FUNCTION_BLOCK FB_RobotComms
VAR
	timWatchDogON: TON;
	timWatchDogOff: TON;
	timMotorsOnFault: TON;
	timMotorsOffFault: TON;
	qMotorsOffFault: BOOL;
	timRunningFault: TON;
	timRunningStopFault: TON;
	tRunRoutine: BOOL;
	timRoutineRunFault: TON;
	tRoutineValMismatch: BOOL;
	timRoutineValMismatchFault: TON;
	qRoutineMismatch: BOOL;
	tRoutineValNotZero: BOOL;
	tRoutineComplete: BOOL;
	tCheckForEndPose: BOOL;
	tCheckForEndPosn: BOOL;
	timFakeRunSignal: TON;
END_VAR

VAR_INPUT
//	iStationPowerOn:BOOL;
//	iStationManualMode:BOOL;
//	iStationAutoCycling:BOOL;
END_VAR
	
VAR_IN_OUT
	iqRobotData:structRobot;
	station:typeStation; //data relating to the entire station
	
END_VAR

VAR_OUTPUT
	qWatchdogFault: BOOL;
	qMotorsOnFault: BOOL;
	qProgramRunFault: BOOL;
	qRoutinePoseFault: BOOL;
	qCollisionFault:BOOL;
END_VAR

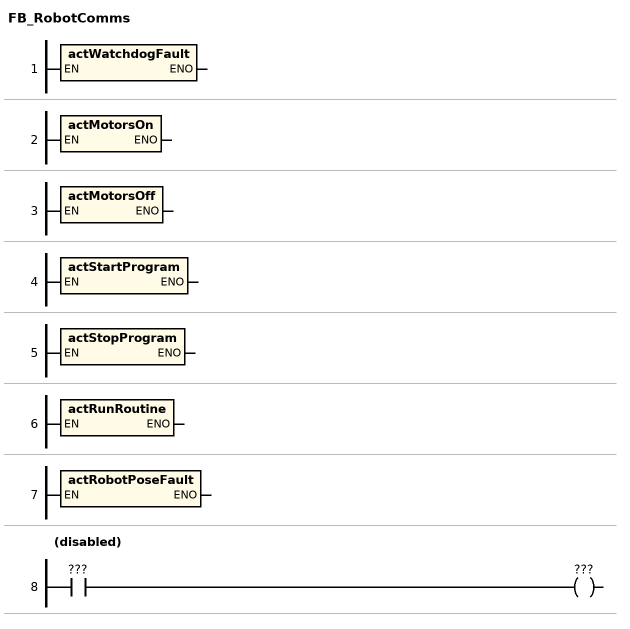
// NETWORK 1
actWatchdogFault();

// NETWORK 2
actMotorsOn();

// NETWORK 3
actMotorsOff();

// NETWORK 4
actStartProgram();

// NETWORK 5
actStopProgram();

// NETWORK 6
actRunRoutine();

// NETWORK 7
actRobotPoseFault();

// NETWORK 8 (disabled)
// ??? := ???;

ACTION actCollision:
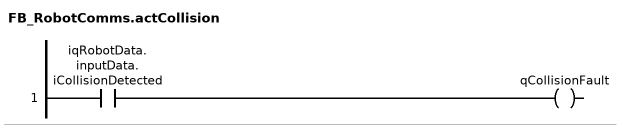
// NETWORK 1
qCollisionFault := iqRobotData.inputData.iCollisionDetected;
END_ACTION

ACTION actMotorsOff:
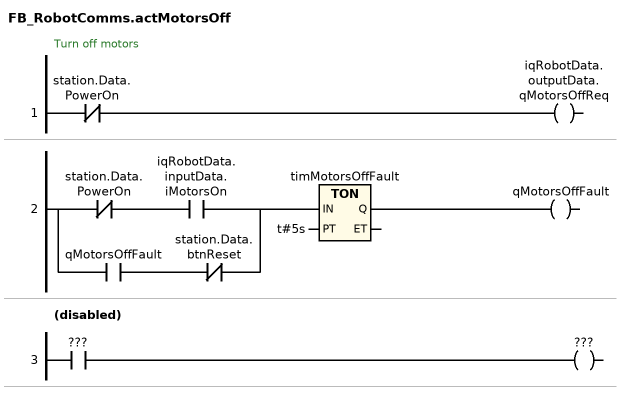
// NETWORK 1
// Turn off motors
iqRobotData.outputData.qMotorsOffReq := NOT station.Data.PowerOn;

// NETWORK 2
timMotorsOffFault(IN := NOT station.Data.PowerOn AND iqRobotData.inputData.iMotorsOn OR qMotorsOffFault AND NOT station.Data.btnReset, PT := t#5s); // TON
qMotorsOffFault := timMotorsOffFault.Q;

// NETWORK 3 (disabled)
// ??? := ???;
END_ACTION

ACTION actMotorsOn:
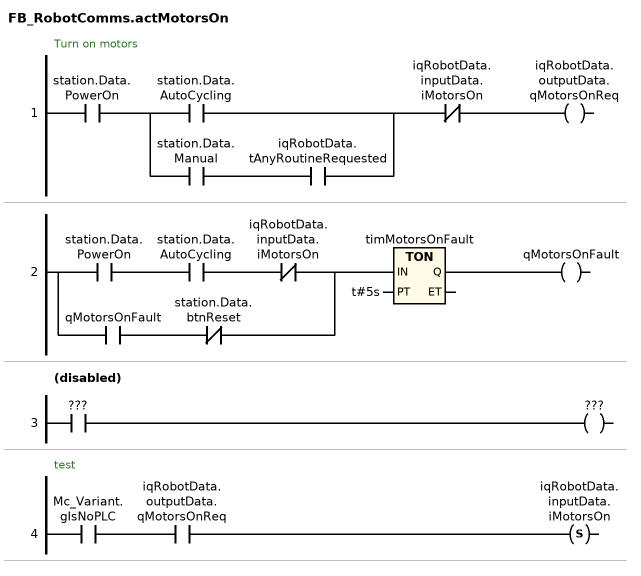
// NETWORK 1
// Turn on motors
iqRobotData.outputData.qMotorsOnReq := station.Data.PowerOn AND (station.Data.AutoCycling OR station.Data.Manual AND iqRobotData.tAnyRoutineRequested) AND NOT iqRobotData.inputData.iMotorsOn;

// NETWORK 2
timMotorsOnFault(IN := station.Data.PowerOn AND station.Data.AutoCycling AND NOT iqRobotData.inputData.iMotorsOn OR qMotorsOnFault AND NOT station.Data.btnReset, PT := t#5s); // TON
qMotorsOnFault := timMotorsOnFault.Q;

// NETWORK 3 (disabled)
// ??? := ???;

// NETWORK 4
// test
iqRobotData.inputData.iMotorsOn S= Mc_Variant.gIsNoPLC AND iqRobotData.outputData.qMotorsOnReq;
END_ACTION

ACTION actRobotPoseFault:
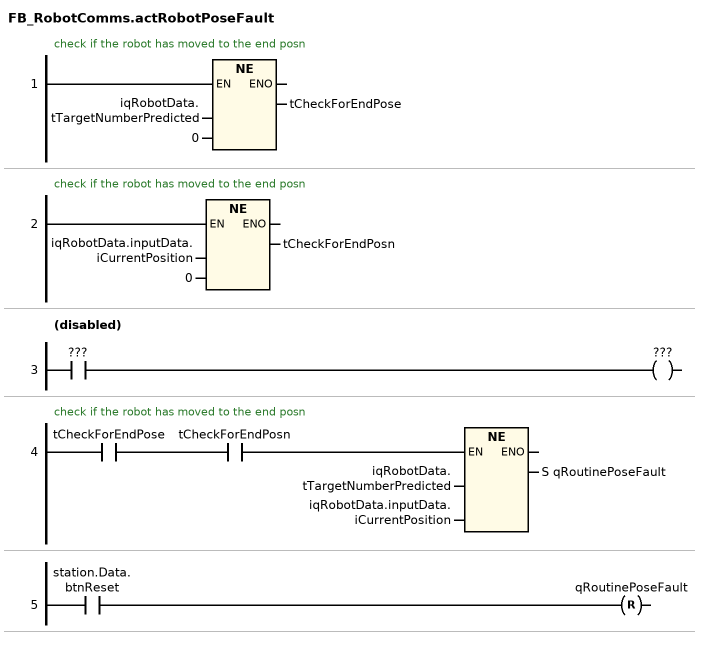
// NETWORK 1
// check if the robot has moved to the end posn
tCheckForEndPose := iqRobotData.tTargetNumberPredicted <> 0;

// NETWORK 2
// check if the robot has moved to the end posn
tCheckForEndPosn := iqRobotData.inputData.iCurrentPosition <> 0;

// NETWORK 3 (disabled)
// ??? := ???;

// NETWORK 4
// check if the robot has moved to the end posn
IF tCheckForEndPose AND tCheckForEndPosn THEN
    qRoutinePoseFault S= iqRobotData.tTargetNumberPredicted <> iqRobotData.inputData.iCurrentPosition;
END_IF

// NETWORK 5
qRoutinePoseFault R= station.Data.btnReset;
END_ACTION

ACTION actRunRoutine:
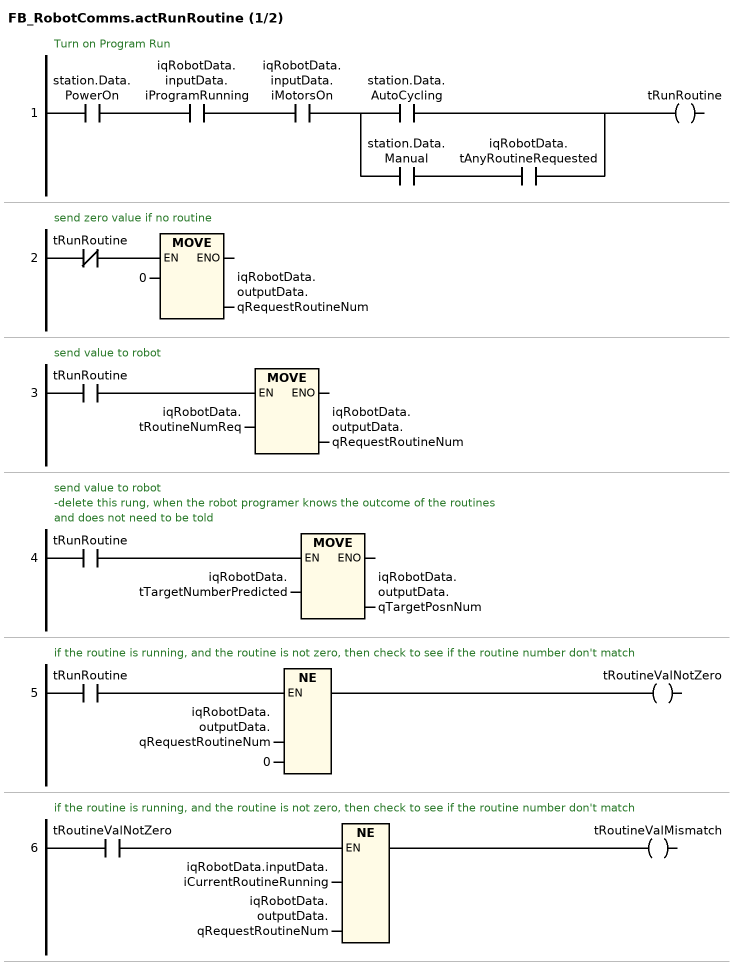
// NETWORK 1
// Turn on Program Run
tRunRoutine := station.Data.PowerOn AND iqRobotData.inputData.iProgramRunning AND iqRobotData.inputData.iMotorsOn AND (station.Data.AutoCycling OR station.Data.Manual AND iqRobotData.tAnyRoutineRequested);

// NETWORK 2
// send zero value if no routine
IF NOT tRunRoutine THEN iqRobotData.outputData.qRequestRoutineNum := 0; END_IF

// NETWORK 3
// send value to robot
IF tRunRoutine THEN iqRobotData.outputData.qRequestRoutineNum := iqRobotData.tRoutineNumReq; END_IF

// NETWORK 4
// send value to robot
// -delete this rung, when the robot programer knows the outcome of the routines
// and does not need to be told
IF tRunRoutine THEN iqRobotData.outputData.qTargetPosnNum := iqRobotData.tTargetNumberPredicted; END_IF

// NETWORK 5
// if the routine is running, and the routine is not zero, then check to see if the routine number don't match
tRoutineValNotZero := tRunRoutine AND iqRobotData.outputData.qRequestRoutineNum <> 0;

// NETWORK 6
// if the routine is running, and the routine is not zero, then check to see if the routine number don't match
tRoutineValMismatch := tRoutineValNotZero AND iqRobotData.inputData.iCurrentRoutineRunning <> iqRobotData.outputData.qRequestRoutineNum;

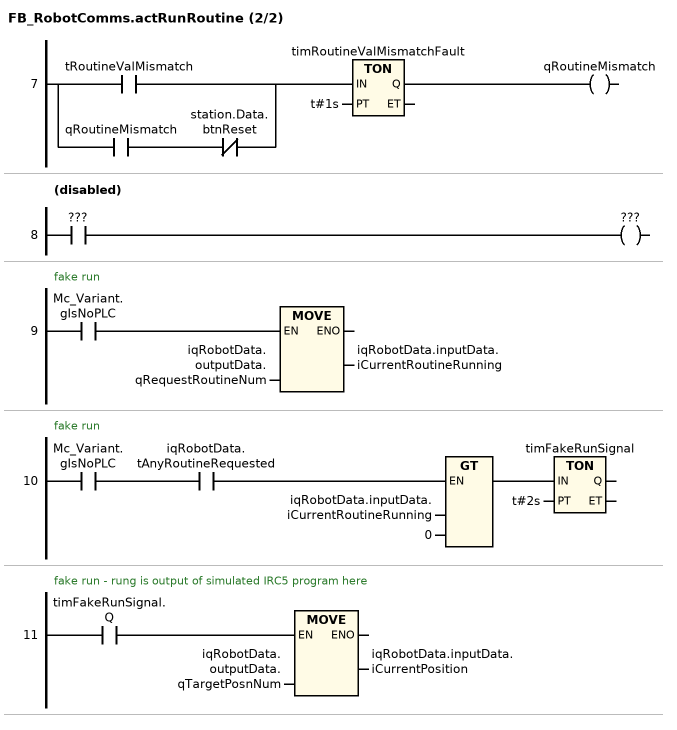
// NETWORK 7
timRoutineValMismatchFault(IN := tRoutineValMismatch OR qRoutineMismatch AND NOT station.Data.btnReset, PT := t#1s); // TON
qRoutineMismatch := timRoutineValMismatchFault.Q;

// NETWORK 8 (disabled)
// ??? := ???;

// NETWORK 9
// fake run
IF Mc_Variant.gIsNoPLC THEN
    iqRobotData.inputData.iCurrentRoutineRunning := iqRobotData.outputData.qRequestRoutineNum;
END_IF

// NETWORK 10
// fake run
timFakeRunSignal(IN := Mc_Variant.gIsNoPLC AND iqRobotData.tAnyRoutineRequested AND iqRobotData.inputData.iCurrentRoutineRunning > 0, PT := t#2s); // TON

// NETWORK 11
// fake run - rung is output of simulated IRC5 program here
IF timFakeRunSignal.Q THEN iqRobotData.inputData.iCurrentPosition := iqRobotData.outputData.qTargetPosnNum; END_IF
END_ACTION

ACTION actStartProgram:
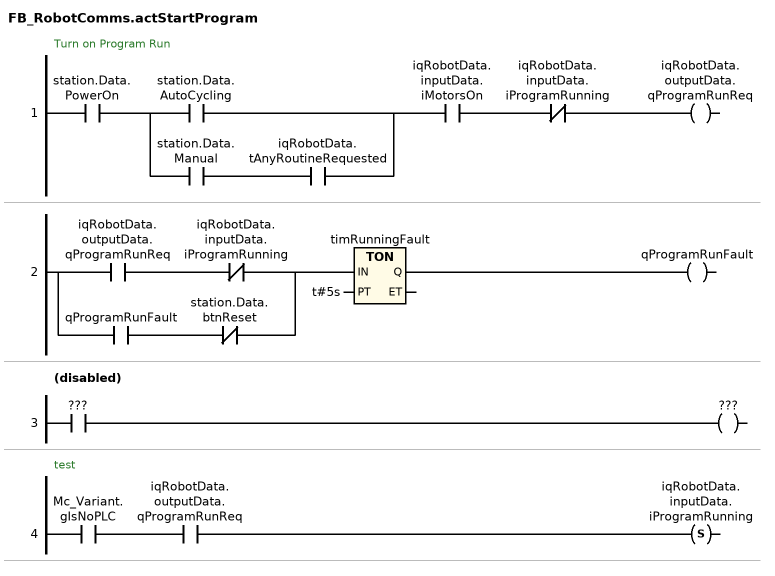
// NETWORK 1
// Turn on Program Run
iqRobotData.outputData.qProgramRunReq := station.Data.PowerOn AND (station.Data.AutoCycling OR station.Data.Manual AND iqRobotData.tAnyRoutineRequested) AND iqRobotData.inputData.iMotorsOn AND NOT iqRobotData.inputData.iProgramRunning;

// NETWORK 2
timRunningFault(IN := iqRobotData.outputData.qProgramRunReq AND NOT iqRobotData.inputData.iProgramRunning OR qProgramRunFault AND NOT station.Data.btnReset, PT := t#5s); // TON
qProgramRunFault := timRunningFault.Q;

// NETWORK 3 (disabled)
// ??? := ???;

// NETWORK 4
// test
iqRobotData.inputData.iProgramRunning S= Mc_Variant.gIsNoPLC AND iqRobotData.outputData.qProgramRunReq;
END_ACTION

ACTION actStopProgram:
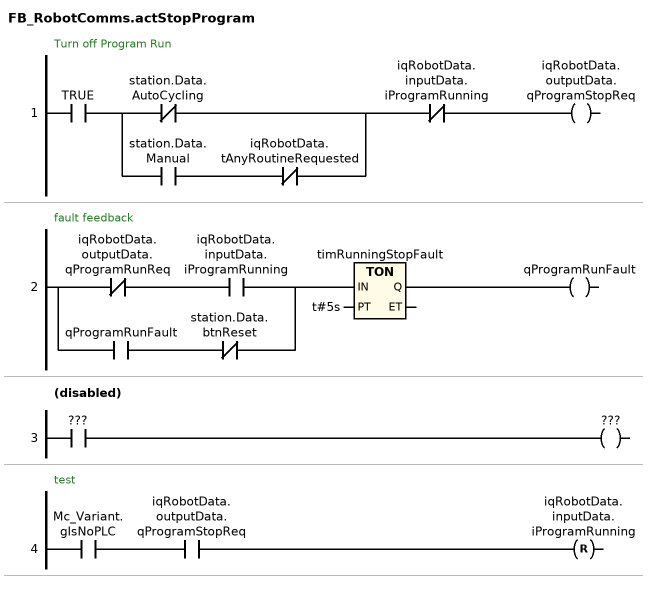
// NETWORK 1
// Turn off Program Run
iqRobotData.outputData.qProgramStopReq := TRUE AND (NOT station.Data.AutoCycling OR station.Data.Manual AND NOT iqRobotData.tAnyRoutineRequested) AND NOT iqRobotData.inputData.iProgramRunning;

// NETWORK 2
// fault feedback
timRunningStopFault(IN := NOT iqRobotData.outputData.qProgramRunReq AND iqRobotData.inputData.iProgramRunning OR qProgramRunFault AND NOT station.Data.btnReset, PT := t#5s); // TON
qProgramRunFault := timRunningStopFault.Q;

// NETWORK 3 (disabled)
// ??? := ???;

// NETWORK 4
// test
iqRobotData.inputData.iProgramRunning R= Mc_Variant.gIsNoPLC AND iqRobotData.outputData.qProgramStopReq;
END_ACTION

ACTION actWatchdogFault:
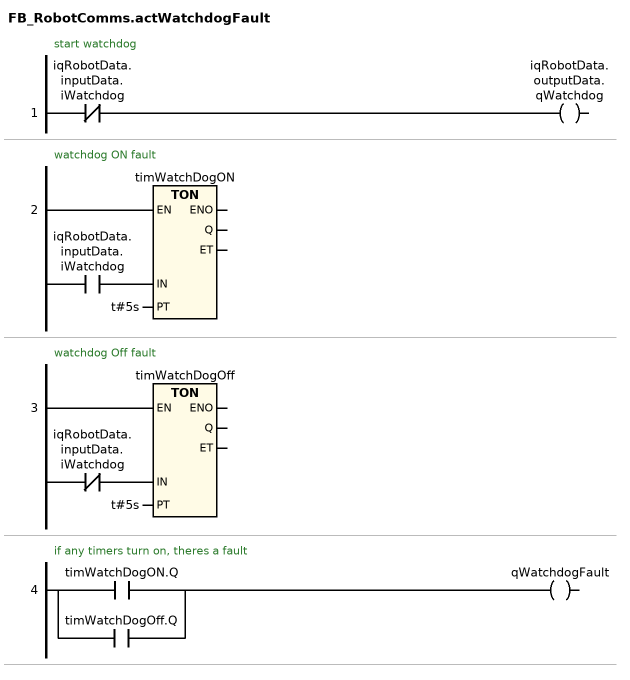
// NETWORK 1
// start watchdog
iqRobotData.outputData.qWatchdog := NOT iqRobotData.inputData.iWatchdog;

// NETWORK 2
// watchdog ON fault
timWatchDogON(IN := iqRobotData.inputData.iWatchdog, PT := t#5s); // TON

// NETWORK 3
// watchdog Off fault
timWatchDogOff(IN := NOT iqRobotData.inputData.iWatchdog, PT := t#5s); // TON

// NETWORK 4
// if any timers turn on, theres a fault
qWatchdogFault := timWatchDogON.Q OR timWatchDogOff.Q;
END_ACTION

END_FUNCTION_BLOCK

(* stored: Version 1.1.0.1, ProductVersion 3.1.4024.11
   POU FB_RobotComms: Id {38d8d4f8-9dcc-4020-a9d8-b9eb8bd54575}, SpecialFunc None
   Action actCollision: Id {ad7d7a71-11d1-4d2a-9400-4cf98c8d3ece}
   Action actMotorsOff: Id {3aae55ed-d4e0-4023-9d06-b2d9a8891dff}
   Action actMotorsOn: Id {95b4a8f2-227b-4515-a580-e1aee86f68f5}
   Action actRobotPoseFault: Id {3d09050b-2fa0-479a-b87f-d5a385822776}
   Action actRunRoutine: Id {d689bbfa-1f33-4904-abbd-05c073ff25b8}
   Action actStartProgram: Id {e94a55d9-064d-4d90-96e9-7cfaead3fb0a}
   Action actStopProgram: Id {c578b1b2-ef79-47a3-b8ec-a48fe2ce8d67}
   Action actWatchdogFault: Id {909cc998-19cb-4223-b55c-ecb0a9ca9da9} *)
